# EPICS substitutions: iocBoot/iocvirPV/virAi.substitutions
file "../../db/virAi.template"{ pattern
{num}
{0}
{1}
{2}
{3}
}
